// TIA Portal project "In OVO done" (V18)

(* hardware
DEVICE "S7-1200 station_1"  S7-1200 Station
   slot 0: "Rack_0"  S7-1200 Rack  Rack  V1.0
   slot 1: "plc1"  CPU 1214C DC/DC/DC  6ES7 214-1AG40-0XB0  V4.6
DEVICE "hmi1"  KTP700 Basic PN
   slot 0: "hmi1"  KTP700 Basic PN  6AV2 123-2GB03-0AX0  17.0.0.0
   slot 1: "HMI_RT_1"  KTP700 Basic PN  6AV2 123-2GB03-0AX0  17.0.0.0
   slot 5: "hmi1.IE_CP_1"  PROFINET Interface  17.0.0.0
      slot 1: "PROFINET Interface_1"  PROFINET Interface
         slot 1: "Port_1"  Port
*)

// ===== PLC "plc1"  CPU 1214C DC/DC/DC =====

VAR_GLOBAL   // PLC tag table "Default tag table"
   "System_Byte" AT %MB1 : Byte;
   "FirstScan" AT %M1.0 : Bool;
   "DiagStatusUpdate" AT %M1.1 : Bool;
   "AlwaysTRUE" AT %M1.2 : Bool;
   "AlwaysFALSE" AT %M1.3 : Bool;
   "Clock_Byte" AT %MB0 : Byte;
   "Clock_10Hz" AT %M0.0 : Bool;
   "Clock_5Hz" AT %M0.1 : Bool;
   "Clock_2.5Hz" AT %M0.2 : Bool;
   "Clock_2Hz" AT %M0.3 : Bool;
   "Clock_1.25Hz" AT %M0.4 : Bool;
   "Clock_1Hz" AT %M0.5 : Bool;
   "Clock_0.625Hz" AT %M0.6 : Bool;
   "Clock_0.5Hz" AT %M0.7 : Bool;
   "Verticaal_hot_end_Pulse" AT %Q980.0 : Bool;
   "Verticaal_hot_end_Direction" AT %Q980.1 : Bool;
END_VAR

VAR_GLOBAL   // PLC tag table "Motor"
   "motorOutput_1" AT %Q981.0 : "stepperMotorOutput";
END_VAR

VAR_GLOBAL   // PLC tag table "Valve"
   "valve1Q" AT %Q980.2 : Bool;
END_VAR

TYPE "stepperMotorInput"
   STRUCT
      axisMove : Bool;
      axisReset : Bool;
      stepOn : Bool;
      jogPlatformDown : Bool;
      jogPlatformUp : Bool;
      stateVerticalStepper : Int;   // 0 = off, 1 = needs initialization, 2 = initializing, 3 = on and initialized
      turnDistance : Real;
      shutOff : Bool;
      motorInitialize : Bool;
      motorInitialized : Bool;
      actualSpeed : Real;
      speedSelector : Int;
   END_STRUCT;
END_TYPE

TYPE "stepperMotorOutput"
   STRUCT
      TO_enable : Bool;
      Step_OFF : Bool;
   END_STRUCT;
END_TYPE

TYPE "stepperMotorSpeed"
   STRUCT
      speed300p : Real := 300.0;
      speed500p : Real := 500.0;
      speed1000p : Real := 1000.0;
      speed2000p : Real := 2000.0;
      speed3000p : Real := 3000.0;
      speed4000p : Real := 4000.0;
      speed5000p : Real := 5000.0;
      speed6000p : Real := 6000.0;
      speed7000p : Real := 7000.0;
      speed8000p : Real := 8000.0;
      speed9000p : Real := 9000.0;
      speed10000p : Real := 10000.0;
      speed11000p : Real := 11000.0;
      speed12000p : Real := 12000.0;
      speed13000p : Real := 13000.0;
      speed14000p : Real := 14000.0;
      speed15000p : Real := 15000.0;
      speed16000p : Real := 16000.0;
      speed17000p : Real := 17000.0;
      speed18000p : Real := 18000.0;
      speed19000p : Real := 19000.0;
      speed20000p : Real := 20000.0;
   END_STRUCT;
END_TYPE

TYPE "valveData"
   STRUCT
      controlHmi : Bool;
      openTime : Time;
      keepOpenHmi : Bool;
   END_STRUCT;
END_TYPE

DATA_BLOCK "openCloseCycle_DB"   // DB19
{ S7_Optimized_Access := 'TRUE' }
VERSION : 0.1
// stored: InstanceOfName openCloseCycle
"openCloseCycle"
BEGIN
END_DATA_BLOCK

DATA_BLOCK "controlStepper_DB"   // DB21
{ S7_Optimized_Access := 'TRUE' }
VERSION : 0.1
// stored: InstanceOfName controlStepper
"controlStepper"
BEGIN
END_DATA_BLOCK

// folder: Stepper/DB's

DATA_BLOCK "initVerticalStepper_DB"   // DB4
{ S7_Optimized_Access := 'TRUE' }
VERSION : 0.1
// stored: InstanceOfName initVerticalStepper
"initVerticalStepper"
BEGIN
END_DATA_BLOCK

DATA_BLOCK "stepperControlDB"   // DB8
{ S7_Optimized_Access := 'TRUE' }
VERSION : 0.1
// stored: InstanceOfName controlStepper
"controlStepper"
BEGIN
END_DATA_BLOCK

DATA_BLOCK "Motor_1"   // DB9
{ S7_Optimized_Access := 'TRUE' }
VERSION : 0.1
   VAR
      motorInput : "stepperMotorInput";
      speedPreSets : "stepperMotorSpeed";
   END_VAR
BEGIN
END_DATA_BLOCK

DATA_BLOCK "moveMotorSpeed_DB"   // DB12
{ S7_Optimized_Access := 'TRUE' }
VERSION : 0.1
// stored: InstanceOfName moveSpeedStepper
"moveSpeedStepper"
BEGIN
END_DATA_BLOCK

DATA_BLOCK "shutOffStepper_DB"   // DB16
{ S7_Optimized_Access := 'TRUE' }
VERSION : 0.1
// stored: InstanceOfName shutOffStepper
"shutOffStepper"
BEGIN
END_DATA_BLOCK

// folder: System blocks/Program resources

DATA_BLOCK "IEC_Timer_0_DB"   // DB1
{ S7_Optimized_Access := 'TRUE' }
AUTHOR : Simatic
FAMILY : IEC
NAME : IEC_TMR
VERSION : 1.0
// stored: InstanceOfName IEC_TIMER
"IEC_TIMER"
BEGIN
END_DATA_BLOCK

DATA_BLOCK "IEC_Timer_0_DB_2"   // DB14
{ S7_Optimized_Access := 'TRUE' }
AUTHOR : Simatic
FAMILY : IEC
NAME : IEC_TMR
VERSION : 1.0
// stored: InstanceOfName IEC_TIMER
"IEC_TIMER"
BEGIN
END_DATA_BLOCK

DATA_BLOCK "IEC_Timer_0_DB_4"   // DB18
{ S7_Optimized_Access := 'TRUE' }
AUTHOR : Simatic
FAMILY : IEC
NAME : IEC_TMR
VERSION : 1.0
// stored: InstanceOfName IEC_TIMER
"IEC_TIMER"
BEGIN
END_DATA_BLOCK

DATA_BLOCK "IEC_Timer_0_DB_8"   // DB24
{ S7_Optimized_Access := 'TRUE' }
AUTHOR : Simatic
FAMILY : IEC
NAME : IEC_TMR
VERSION : 1.0
// stored: InstanceOfName IEC_TIMER
"IEC_TIMER"
BEGIN
END_DATA_BLOCK

// folder: Valves/DB's

DATA_BLOCK "valvesDB"   // DB17
{ S7_Optimized_Access := 'TRUE' }
VERSION : 0.1
   VAR
      valve1 : "valveData";
   END_VAR
BEGIN
   valve1.openTime := T#500ms;
END_DATA_BLOCK

// folder: (top level)

DATA_BLOCK "VerticalHotEnd"   // DB2, Motion_DB
{ S7_Optimized_Access := 'TRUE' }
AUTHOR : SIMATIC
FAMILY : BasicMC
NAME : TO_PosAx
VERSION : 8.0
// stored: InstanceOfName TO_PositioningAxis
"TO_PositioningAxis"
BEGIN
   // Axis.EnableOutput_AddressCU = %Q981.0
   // Axis.DirectionOutputEnabledCU = TRUE
   // Axis.LengthUnit.LastDistance = -1
   // Axis.OnlinePtoModeCU = 16#0000_0002
   // Axis.SelectedChannel2EnumCU = %Q980.1
   // Axis.SelectedChannel1EnumCU = %Q980.0
   // Pulse.MinDeltaDeltaFrequencyCU = 0.004
   // Pulse.MaxDeltaDeltaFrequencyCU = 1.0E+10
   // Pulse.MinDeltaFrequencyCU = 0.005
   // Pulse.MaxDeltaFrequencyCU = 9.5E+9
   // Pulse.MinFrequencyCU = 1.0
   // Pulse.MaxFrequencyCU = 100000.0
   // Pulse.OutputSourceCU = 16#0000_0000
   // Axis.SelectPTO = 0
END_DATA_BLOCK

ORGANIZATION_BLOCK "Main"   // OB1, LAD, ProgramCycle
TITLE = "Main Program Sweep (Cycle)"
{ S7_Optimized_Access := 'TRUE' }
VERSION : 0.1
   VAR_INPUT
      Initial_Call : Bool;   // Initial call of this OB
      Remanence : Bool;   // =True, if remanent data are available
   END_VAR
BEGIN

REGION Network 1: If state is 0 but stepOn is True then change state to 1
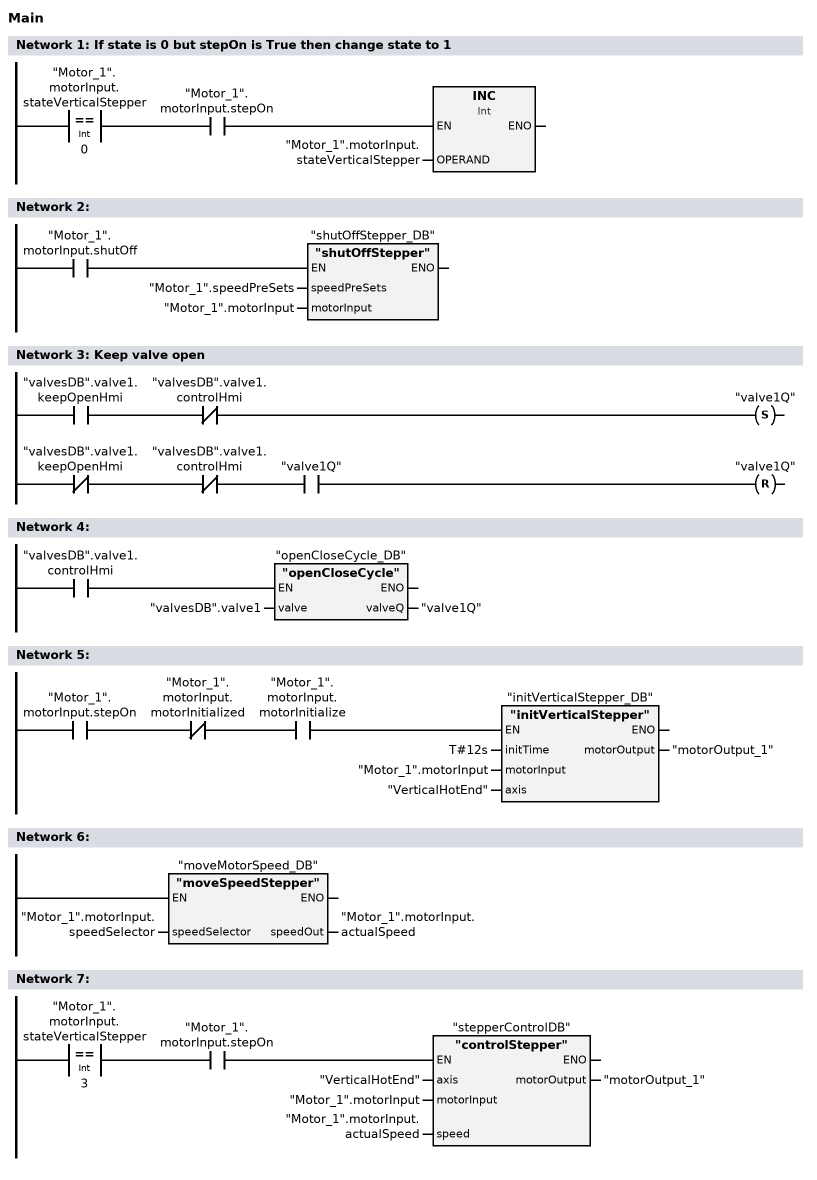
   RUNG wire#powerrail
      { S7_Templates := "SrcType := Int" } EQ_Contact(in1 := "Motor_1".motorInput.stateVerticalStepper, in2 := 0)
      Contact( "Motor_1".motorInput.stepOn )
      { S7_Templates := "DestType := Int" } Inc( "Motor_1".motorInput.stateVerticalStepper )
   END_RUNG
   // the same network as SCL:
   IF ("Motor_1".motorInput.stateVerticalStepper = 0) AND "Motor_1".motorInput.stepOn THEN
       "Motor_1".motorInput.stateVerticalStepper := "Motor_1".motorInput.stateVerticalStepper + 1;
   END_IF;
END_REGION

REGION Network 2
   RUNG wire#powerrail
      Contact( "Motor_1".motorInput.shutOff )
      "shutOffStepper_DB"(speedPreSets := "Motor_1".speedPreSets, motorInput := "Motor_1".motorInput)
   END_RUNG
   // the same network as SCL:
   IF "Motor_1".motorInput.shutOff THEN
       "shutOffStepper_DB"(speedPreSets := "Motor_1".speedPreSets, motorInput := "Motor_1".motorInput);   // "shutOffStepper"
   END_IF;
END_REGION

REGION Network 3: Keep valve open
   RUNG wire#powerrail
      Contact( "valvesDB".valve1.keepOpenHmi )
      I_Contact( "valvesDB".valve1.controlHmi )
      S_Coil( "valve1Q" )
   END_RUNG
   RUNG wire#powerrail
      I_Contact( "valvesDB".valve1.keepOpenHmi )
      I_Contact( "valvesDB".valve1.controlHmi )
      Contact( "valve1Q" )
      R_Coil( "valve1Q" )
   END_RUNG
   // the same network as SCL:
   IF "valvesDB".valve1.keepOpenHmi AND NOT "valvesDB".valve1.controlHmi THEN "valve1Q" := TRUE; END_IF;
   IF NOT "valvesDB".valve1.keepOpenHmi AND NOT "valvesDB".valve1.controlHmi AND "valve1Q" THEN
       "valve1Q" := FALSE;
   END_IF;
END_REGION

REGION Network 4
   RUNG wire#powerrail
      Contact( "valvesDB".valve1.controlHmi )
      "openCloseCycle_DB"(valve := "valvesDB".valve1, valveQ => "valve1Q")
   END_RUNG
   // the same network as SCL:
   IF "valvesDB".valve1.controlHmi THEN
       "openCloseCycle_DB"(valve := "valvesDB".valve1, valveQ => "valve1Q");   // "openCloseCycle"
   END_IF;
END_REGION

REGION Network 5
   RUNG wire#powerrail
      Contact( "Motor_1".motorInput.stepOn )
      I_Contact( "Motor_1".motorInput.motorInitialized )
      Contact( "Motor_1".motorInput.motorInitialize )
      "initVerticalStepper_DB"(initTime := T#12s, motorInput := "Motor_1".motorInput, axis := "VerticalHotEnd", motorOutput => "motorOutput_1")
   END_RUNG
   // the same network as SCL:
   IF "Motor_1".motorInput.stepOn AND NOT "Motor_1".motorInput.motorInitialized AND "Motor_1".motorInput.motorInitialize THEN
       "initVerticalStepper_DB"(initTime := T#12s,   // "initVerticalStepper"
                               motorInput := "Motor_1".motorInput,
                               axis := "VerticalHotEnd",
                               motorOutput => "motorOutput_1");
   END_IF;
END_REGION

REGION Network 6
   RUNG wire#powerrail
      "moveMotorSpeed_DB"(speedSelector := "Motor_1".motorInput.speedSelector, speedOut => "Motor_1".motorInput.actualSpeed)
   END_RUNG
   // the same network as SCL:
   "moveMotorSpeed_DB"(speedSelector := "Motor_1".motorInput.speedSelector,   // "moveSpeedStepper"
                       speedOut => "Motor_1".motorInput.actualSpeed);
END_REGION

REGION Network 7
   RUNG wire#powerrail
      { S7_Templates := "SrcType := Int" } EQ_Contact(in1 := "Motor_1".motorInput.stateVerticalStepper, in2 := 3)
      Contact( "Motor_1".motorInput.stepOn )
      "stepperControlDB"(axis := "VerticalHotEnd", motorInput := "Motor_1".motorInput, speed := "Motor_1".motorInput.actualSpeed, motorOutput => "motorOutput_1")
   END_RUNG
   // the same network as SCL:
   IF ("Motor_1".motorInput.stateVerticalStepper = 3) AND "Motor_1".motorInput.stepOn THEN
       "stepperControlDB"(axis := "VerticalHotEnd",   // "controlStepper"
                          motorInput := "Motor_1".motorInput,
                          speed := "Motor_1".motorInput.actualSpeed,
                          motorOutput => "motorOutput_1");
   END_IF;
END_REGION
END_ORGANIZATION_BLOCK

// folder: Stepper

FUNCTION_BLOCK "controlStepper"   // FB1, LAD
{ S7_Optimized_Access := 'TRUE' }
VERSION : 0.1
   VAR_INPUT
      axis : TO_PositioningAxis;
      motorInput : "stepperMotorInput";
      speed : Int;
   END_VAR
   VAR_OUTPUT
      motorOutput : "stepperMotorOutput";
   END_VAR
BEGIN

REGION Network 1: enable motor
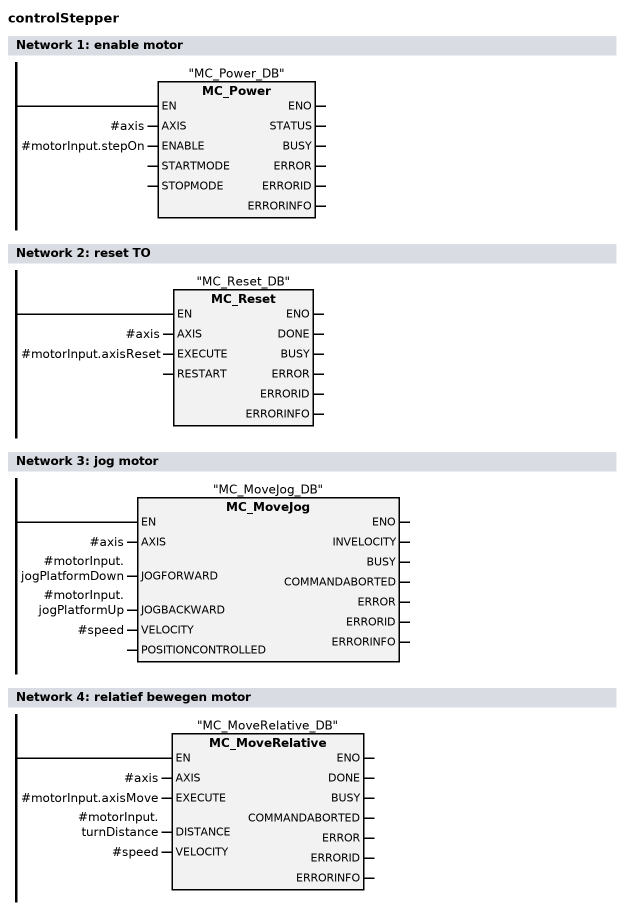
   "MC_Power_DB"(Axis := #axis, Enable := #motorInput.stepOn);   // MC_Power
END_REGION

REGION Network 2: reset TO
   "MC_Reset_DB"(Axis := #axis, Execute := #motorInput.axisReset);   // MC_Reset
END_REGION

REGION Network 3: jog motor
   "MC_MoveJog_DB"(Axis := #axis,   // MC_MoveJog
                   JogForward := #motorInput.jogPlatformDown,
                   JogBackward := #motorInput.jogPlatformUp,
                   Velocity := #speed);
END_REGION

REGION Network 4: relatief bewegen motor
   "MC_MoveRelative_DB"(Axis := #axis,   // MC_MoveRelative
                        Execute := #motorInput.axisMove,
                        Distance := #motorInput.turnDistance,
                        Velocity := #speed);
END_REGION
END_FUNCTION_BLOCK

FUNCTION_BLOCK "initVerticalStepper"   // FB2, LAD
TITLE = Initialize vertical stepper
{ S7_Optimized_Access := 'TRUE' }
VERSION : 0.1
   VAR_INPUT
      initTime : Time;
   END_VAR
   VAR_OUTPUT
      motorOutput : "stepperMotorOutput";
   END_VAR
   VAR_IN_OUT
      motorInput : "stepperMotorInput";
      axis : TO_PositioningAxis;
   END_VAR
BEGIN

REGION Network 1: Turn platform into screw thread and set state to initializing. Set a timer and after that reset the initialize tag and set state to "on and initialized"
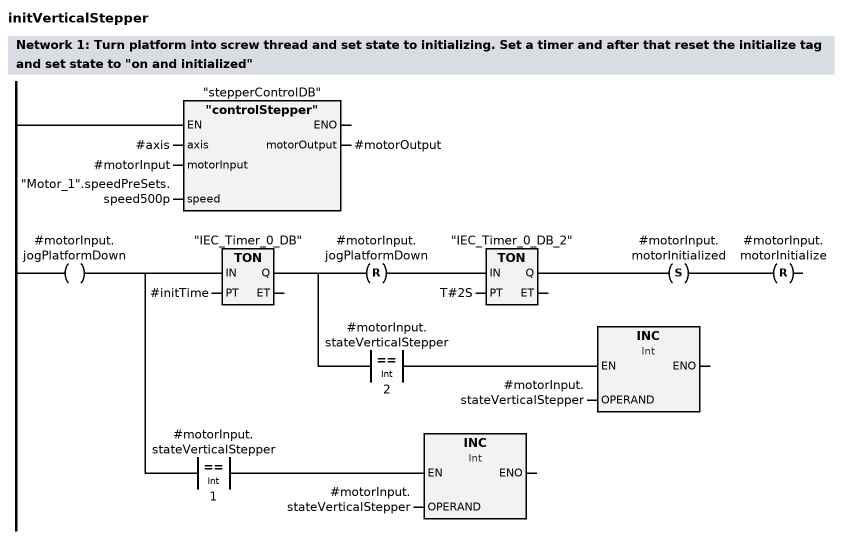
   "stepperControlDB"(axis := #axis,   // "controlStepper"
                      motorInput := #motorInput,
                      speed := "Motor_1".speedPreSets.speed500p,
                      motorOutput => #motorOutput);
   #motorInput.jogPlatformDown := TRUE;
   "IEC_Timer_0_DB".TON(IN := TRUE, PT := #initTime);
   IF "IEC_Timer_0_DB".Q THEN #motorInput.jogPlatformDown := FALSE; END_IF;
   "IEC_Timer_0_DB_2".TON(IN := "IEC_Timer_0_DB".Q, PT := T#2S);
   IF "IEC_Timer_0_DB_2".Q THEN
       #motorInput.motorInitialized := TRUE;
       #motorInput.motorInitialize := FALSE;
   END_IF;
   IF "IEC_Timer_0_DB".Q AND (#motorInput.stateVerticalStepper = 2) THEN
       #motorInput.stateVerticalStepper := #motorInput.stateVerticalStepper + 1;
   END_IF;
   IF #motorInput.stateVerticalStepper = 1 THEN
       #motorInput.stateVerticalStepper := #motorInput.stateVerticalStepper + 1;
   END_IF;
END_REGION
END_FUNCTION_BLOCK

FUNCTION_BLOCK "moveSpeedStepper"   // FB4, LAD
{ S7_Optimized_Access := 'TRUE' }
VERSION : 0.1
   VAR_INPUT
      speedSelector : Int;
   END_VAR
   VAR_OUTPUT
      speedOut : Real;
   END_VAR
   VAR
      speeds : "stepperMotorSpeed";
   END_VAR
BEGIN

REGION Network 1
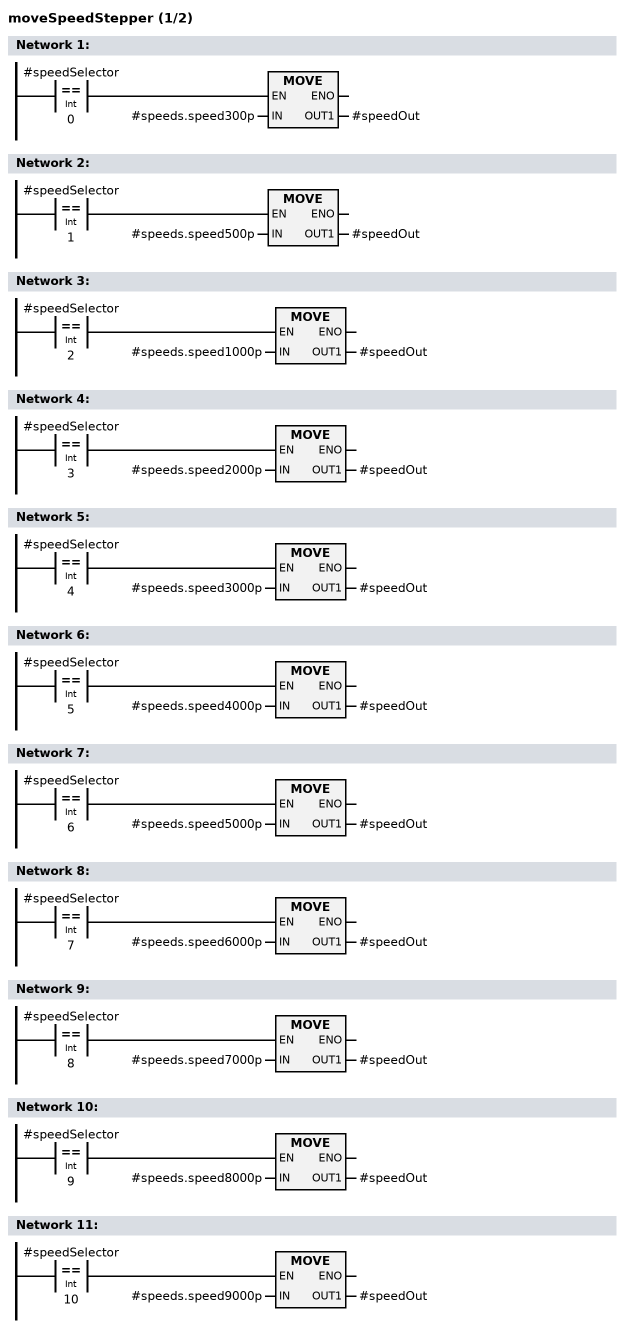
   RUNG wire#powerrail
      { S7_Templates := "SrcType := Int" } EQ_Contact(in1 := #speedSelector, in2 := 0)
      Move(in := #speeds.speed300p, out1 => #speedOut)
   END_RUNG
   // the same network as SCL:
   IF #speedSelector = 0 THEN #speedOut := #speeds.speed300p; END_IF;
END_REGION

REGION Network 2
   RUNG wire#powerrail
      { S7_Templates := "SrcType := Int" } EQ_Contact(in1 := #speedSelector, in2 := 1)
      Move(in := #speeds.speed500p, out1 => #speedOut)
   END_RUNG
   // the same network as SCL:
   IF #speedSelector = 1 THEN #speedOut := #speeds.speed500p; END_IF;
END_REGION

REGION Network 3
   RUNG wire#powerrail
      { S7_Templates := "SrcType := Int" } EQ_Contact(in1 := #speedSelector, in2 := 2)
      Move(in := #speeds.speed1000p, out1 => #speedOut)
   END_RUNG
   // the same network as SCL:
   IF #speedSelector = 2 THEN #speedOut := #speeds.speed1000p; END_IF;
END_REGION

REGION Network 4
   RUNG wire#powerrail
      { S7_Templates := "SrcType := Int" } EQ_Contact(in1 := #speedSelector, in2 := 3)
      Move(in := #speeds.speed2000p, out1 => #speedOut)
   END_RUNG
   // the same network as SCL:
   IF #speedSelector = 3 THEN #speedOut := #speeds.speed2000p; END_IF;
END_REGION

REGION Network 5
   RUNG wire#powerrail
      { S7_Templates := "SrcType := Int" } EQ_Contact(in1 := #speedSelector, in2 := 4)
      Move(in := #speeds.speed3000p, out1 => #speedOut)
   END_RUNG
   // the same network as SCL:
   IF #speedSelector = 4 THEN #speedOut := #speeds.speed3000p; END_IF;
END_REGION

REGION Network 6
   RUNG wire#powerrail
      { S7_Templates := "SrcType := Int" } EQ_Contact(in1 := #speedSelector, in2 := 5)
      Move(in := #speeds.speed4000p, out1 => #speedOut)
   END_RUNG
   // the same network as SCL:
   IF #speedSelector = 5 THEN #speedOut := #speeds.speed4000p; END_IF;
END_REGION

REGION Network 7
   RUNG wire#powerrail
      { S7_Templates := "SrcType := Int" } EQ_Contact(in1 := #speedSelector, in2 := 6)
      Move(in := #speeds.speed5000p, out1 => #speedOut)
   END_RUNG
   // the same network as SCL:
   IF #speedSelector = 6 THEN #speedOut := #speeds.speed5000p; END_IF;
END_REGION

REGION Network 8
   RUNG wire#powerrail
      { S7_Templates := "SrcType := Int" } EQ_Contact(in1 := #speedSelector, in2 := 7)
      Move(in := #speeds.speed6000p, out1 => #speedOut)
   END_RUNG
   // the same network as SCL:
   IF #speedSelector = 7 THEN #speedOut := #speeds.speed6000p; END_IF;
END_REGION

REGION Network 9
   RUNG wire#powerrail
      { S7_Templates := "SrcType := Int" } EQ_Contact(in1 := #speedSelector, in2 := 8)
      Move(in := #speeds.speed7000p, out1 => #speedOut)
   END_RUNG
   // the same network as SCL:
   IF #speedSelector = 8 THEN #speedOut := #speeds.speed7000p; END_IF;
END_REGION

REGION Network 10
   RUNG wire#powerrail
      { S7_Templates := "SrcType := Int" } EQ_Contact(in1 := #speedSelector, in2 := 9)
      Move(in := #speeds.speed8000p, out1 => #speedOut)
   END_RUNG
   // the same network as SCL:
   IF #speedSelector = 9 THEN #speedOut := #speeds.speed8000p; END_IF;
END_REGION

REGION Network 11
   RUNG wire#powerrail
      { S7_Templates := "SrcType := Int" } EQ_Contact(in1 := #speedSelector, in2 := 10)
      Move(in := #speeds.speed9000p, out1 => #speedOut)
   END_RUNG
   // the same network as SCL:
   IF #speedSelector = 10 THEN #speedOut := #speeds.speed9000p; END_IF;
END_REGION

REGION Network 12
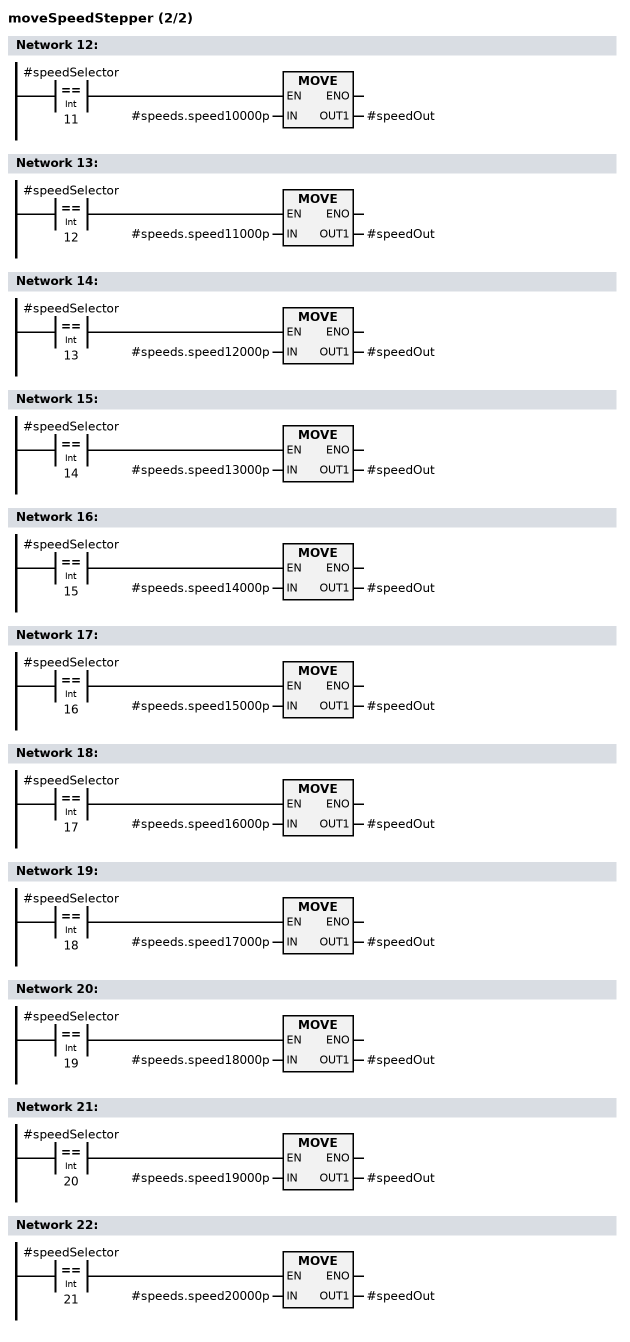
   RUNG wire#powerrail
      { S7_Templates := "SrcType := Int" } EQ_Contact(in1 := #speedSelector, in2 := 11)
      Move(in := #speeds.speed10000p, out1 => #speedOut)
   END_RUNG
   // the same network as SCL:
   IF #speedSelector = 11 THEN #speedOut := #speeds.speed10000p; END_IF;
END_REGION

REGION Network 13
   RUNG wire#powerrail
      { S7_Templates := "SrcType := Int" } EQ_Contact(in1 := #speedSelector, in2 := 12)
      Move(in := #speeds.speed11000p, out1 => #speedOut)
   END_RUNG
   // the same network as SCL:
   IF #speedSelector = 12 THEN #speedOut := #speeds.speed11000p; END_IF;
END_REGION

REGION Network 14
   RUNG wire#powerrail
      { S7_Templates := "SrcType := Int" } EQ_Contact(in1 := #speedSelector, in2 := 13)
      Move(in := #speeds.speed12000p, out1 => #speedOut)
   END_RUNG
   // the same network as SCL:
   IF #speedSelector = 13 THEN #speedOut := #speeds.speed12000p; END_IF;
END_REGION

REGION Network 15
   RUNG wire#powerrail
      { S7_Templates := "SrcType := Int" } EQ_Contact(in1 := #speedSelector, in2 := 14)
      Move(in := #speeds.speed13000p, out1 => #speedOut)
   END_RUNG
   // the same network as SCL:
   IF #speedSelector = 14 THEN #speedOut := #speeds.speed13000p; END_IF;
END_REGION

REGION Network 16
   RUNG wire#powerrail
      { S7_Templates := "SrcType := Int" } EQ_Contact(in1 := #speedSelector, in2 := 15)
      Move(in := #speeds.speed14000p, out1 => #speedOut)
   END_RUNG
   // the same network as SCL:
   IF #speedSelector = 15 THEN #speedOut := #speeds.speed14000p; END_IF;
END_REGION

REGION Network 17
   RUNG wire#powerrail
      { S7_Templates := "SrcType := Int" } EQ_Contact(in1 := #speedSelector, in2 := 16)
      Move(in := #speeds.speed15000p, out1 => #speedOut)
   END_RUNG
   // the same network as SCL:
   IF #speedSelector = 16 THEN #speedOut := #speeds.speed15000p; END_IF;
END_REGION

REGION Network 18
   RUNG wire#powerrail
      { S7_Templates := "SrcType := Int" } EQ_Contact(in1 := #speedSelector, in2 := 17)
      Move(in := #speeds.speed16000p, out1 => #speedOut)
   END_RUNG
   // the same network as SCL:
   IF #speedSelector = 17 THEN #speedOut := #speeds.speed16000p; END_IF;
END_REGION

REGION Network 19
   RUNG wire#powerrail
      { S7_Templates := "SrcType := Int" } EQ_Contact(in1 := #speedSelector, in2 := 18)
      Move(in := #speeds.speed17000p, out1 => #speedOut)
   END_RUNG
   // the same network as SCL:
   IF #speedSelector = 18 THEN #speedOut := #speeds.speed17000p; END_IF;
END_REGION

REGION Network 20
   RUNG wire#powerrail
      { S7_Templates := "SrcType := Int" } EQ_Contact(in1 := #speedSelector, in2 := 19)
      Move(in := #speeds.speed18000p, out1 => #speedOut)
   END_RUNG
   // the same network as SCL:
   IF #speedSelector = 19 THEN #speedOut := #speeds.speed18000p; END_IF;
END_REGION

REGION Network 21
   RUNG wire#powerrail
      { S7_Templates := "SrcType := Int" } EQ_Contact(in1 := #speedSelector, in2 := 20)
      Move(in := #speeds.speed19000p, out1 => #speedOut)
   END_RUNG
   // the same network as SCL:
   IF #speedSelector = 20 THEN #speedOut := #speeds.speed19000p; END_IF;
END_REGION

REGION Network 22
   RUNG wire#powerrail
      { S7_Templates := "SrcType := Int" } EQ_Contact(in1 := #speedSelector, in2 := 21)
      Move(in := #speeds.speed20000p, out1 => #speedOut)
   END_RUNG
   // the same network as SCL:
   IF #speedSelector = 21 THEN #speedOut := #speeds.speed20000p; END_IF;
END_REGION
END_FUNCTION_BLOCK

FUNCTION_BLOCK "shutOffStepper"   // FB5, LAD
{ S7_Optimized_Access := 'TRUE' }
VERSION : 0.1
   VAR_INPUT
      speedPreSets : "stepperMotorSpeed";
   END_VAR
   VAR_IN_OUT
      motorInput : "stepperMotorInput";
   END_VAR
BEGIN

REGION Network 1
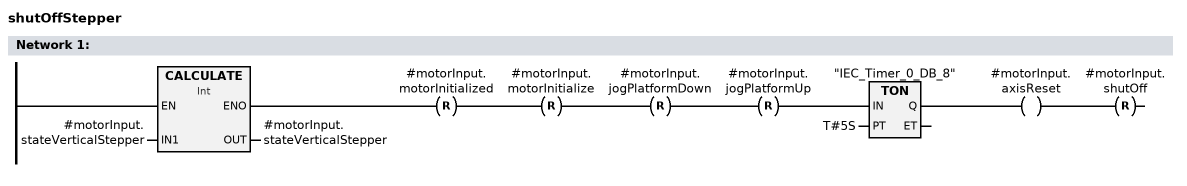
   #motorInput.stateVerticalStepper := #motorInput.stateVerticalStepper-#motorInput.stateVerticalStepper;
   #motorInput.motorInitialized := FALSE;
   #motorInput.motorInitialize := FALSE;
   #motorInput.jogPlatformDown := FALSE;
   #motorInput.jogPlatformUp := FALSE;
   "IEC_Timer_0_DB_8".TON(IN := TRUE, PT := T#5S);
   #motorInput.axisReset := "IEC_Timer_0_DB_8".Q;
   IF "IEC_Timer_0_DB_8".Q THEN #motorInput.shutOff := FALSE; END_IF;
END_REGION
END_FUNCTION_BLOCK

// folder: Valves

FUNCTION_BLOCK "openCloseCycle"   // FB7, LAD
{ S7_Optimized_Access := 'TRUE' }
VERSION : 0.1
   VAR_OUTPUT
      valveQ : Bool;
   END_VAR
   VAR_IN_OUT
      valve : "valveData";
   END_VAR
   VAR_TEMP   // added for the SCL form of the ladder/FBD networks
      _w1 : Bool;
   END_VAR
BEGIN

REGION Network 1
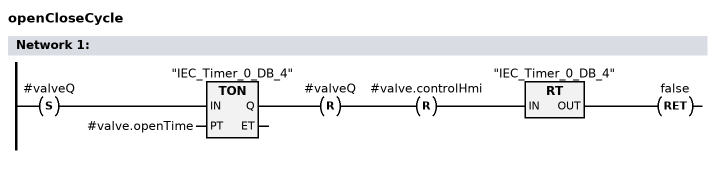
   #valveQ := TRUE;
   "IEC_Timer_0_DB_4".TON(IN := TRUE, PT := #valve.openTime);
   IF "IEC_Timer_0_DB_4".Q THEN
       #valveQ := FALSE;
       #valve.controlHmi := FALSE;
   END_IF;
   #_w1 := "IEC_Timer_0_DB_4".Q;
   IF #_w1 THEN
       RESET_TIMER("IEC_Timer_0_DB_4");
       ENO := false;
       RETURN;
   END_IF;
END_REGION
END_FUNCTION_BLOCK

(* ===== HMI "HMI_RT_1" =====
system functions are stored by id; their names below are inferred from use
connection "HMI_Connection_1": ETHERNET, SMART_S7_1200_OMS

HMI tags "Default tag table"
   "Tag_ScreenNumber" : UInt, internal
   "valveEggs_1" : Bool = PLC valve1Q AT %Q980.2, 100 ms
   "valvesDB_valve1_controlHmi" : Bool = PLC valvesDB.valve1.controlHmi, 100 ms
   "valvesDB_valve1_openTime" : Time = PLC valvesDB.valve1.openTime, 100 ms
   "valvesDB_valve1_keepOpenHmi" : Bool = PLC valvesDB.valve1.keepOpenHmi, 100 ms

HMI tags "Stepper_motor"
   "Motor_Q_1" : stepperMotorOutput = PLC motorOutput_1 AT %Q981.0, 100 ms
   "Motor_I_1" : stepperMotorInput = PLC Motor_1.motorInput AT %DB1.DBW0, 100 ms
   "Verticaal_hot_end_Direction" : Bool = PLC Verticaal_hot_end_Direction AT %Q980.1, 1 s
   "Verticaal_hot_end_Pulse" : Bool = PLC Verticaal_hot_end_Pulse AT %Q980.0, 1 s

Template "Template_1" 800x480
   Button "Template_Button_3" at 316,429 size 71x50; TextOff 'Text'
   Button "Exit" at 714,429 size 71x50; TextOff 'Exit'; PictureOff "ExitRuntime_KTP700_Basic_PN_TR"; PictureOn "ExitRuntime_KTP700_Basic_PN_TR"
      on Release: StopRuntime(0)
   Button "Template_Button" at 614,429 size 71x50; TextOff 'Text'
   Button "Template_Button_1" at 514,429 size 71x50; TextOff 'Text'
   Button "Template_Button_2" at 414,429 size 71x50; TextOff 'Text'
   Button "Template_Button_4" at 214,429 size 71x50; TextOff 'Text'
   Button "Alarms" at 114,429 size 71x50; TextOff 'Alarms'; PictureOff "AlarmDisplay_KTP700_Basic_PN_TR"; PictureOn "AlarmDisplay_KTP700_Basic_PN_TR"
      on Release: function_ef3f5d25("Alarm window_Unacknowledged", -1)
   Button "Start screen" at 14,429 size 71x50; TextOff 'Start screen'; PictureOff "NavigateHome_KTP700_Basic_PN_TR"; PictureOn "NavigateHome_KTP700_Basic_PN_TR"
      on Release: ActivateScreen("Root screen", 0)
   SymbolicIOField "Symbolic_IO_Field_Screen" at 93,9 size 600x33; TextOff '0'; TextOn '1'; TextList "TextList_ScreenNames"
      ProcessValue <- "Tag_ScreenNumber"
      on Change: ActivateScreenByNumber("Tag_ScreenNumber", 0)
   DateTimeField "HmiScreenItemData" at 695,25 size 105x25
   DateTimeField "HmiScreenItemData_1" at 695,0 size 105x25
   GraphicView "Logo" at 0,0 size 91x51; Picture "In+Ovo+logo_2"

screen "Root screen" 800x480, template "Template_1"
   on GenerateScreen: SetTag("Tag_ScreenNumber", 1)
   Button "Button_3" at 404,264 size 148x64; TextOff 'Start glueing'; PictureOff "Graphic_2"
      on Press: SetBit("valvesDB_valve1_controlHmi"); ResetBit("valvesDB_valve1_keepOpenHmi"); function_b14e0dd5("valvesDB_valve1_controlHmi", 0)
   GraphicView "Graphic view_1" at 334,141 size 133x70; Picture "Graphic_1"
   TextField "Text field_1" at 302,107 size 197x23; Text 'Vertical stepper motors'
   Circle "Circle_1" at 445,224 size 32x32
      Appearance <- "stateVerticalStepper"
   Switch "Switch_1" at 329,224 size 109x32; CaptionText 'Switch'; TextOff 'OFF'; TextOn 'ON'
      ProcessValue <- "stepOn"
      on SwitchOff: SetBit("shutOff")
   Button "Button_1" at 245,264 size 148x64; TextOff 'Initialize'
      on Press: SetBit("motorInitialize")
   Button "Button_2" at 245,336 size 307x32; TextOff 'Manual control/settings'; TextOn 'Manual control'
      on Click: ActivateScreen("Manual control", 0)
   GraphicView "Graphic view_2" at 570,118 size 183x250; Picture "580b57fbd9996e24bc43c108"
   GraphicView "Graphic view_3" at 18,129 size 225x239; Picture "308-3089671_baby-chicken-free-png-image-chick-transparent-png"

screen "Manual control" 800x480, template "Template_1"
   Button "Button_2" at 226,210 size 109x64; TextOff 'Down'
      on Release: ResetBit("jogPlatformDown")
      on Press: SetBit("jogPlatformDown"); ResetBit("jogPlatformUp")
   Button "Button_3" at 226,136 size 109x64; TextOff 'Up'
      on Release: ResetBit("jogPlatformUp")
      on Press: SetBit("jogPlatformUp"); ResetBit("jogPlatformDown")
   IOField "I/O field_1" at 593,168 size 109x32; FormatPattern s999999999.999
      ProcessValue <- "turnDistance"
   Button "Button_4" at 227,284 size 109x64; TextOff 'Move'
      on Release: ResetBit("axisMove")
      on Press: SetBit("axisMove")
   TextField "Text field_3" at 238,105 size 86x23; Text 'Jog/move'
   TextField "Text field_4" at 345,105 size 112x23; Text 'Valve control'
   TextField "Text field_2" at 587,136 size 121x23; Text 'Move distance'
   IOField "I/O field_2" at 593,242 size 109x32; FormatPattern s999999999.999
      ProcessValue <- "actualSpeed"
   Button "Button_5" at 466,136 size 109x64; TextOff '+'; PictureOff "Graphic_2"
      on Press: function_dd21b452("speedSelector", 1)
   Button "Button_6" at 466,210 size 109x64; TextOff '-'; PictureOff "Graphic_3"
      on Press: function_b9b71300("speedSelector", 1)
   TextField "Text field_5" at 593,210 size 109x32; Text 'Jog speed'
   Button "Button_1" at 226,359 size 349x32; TextOff 'Root screen'
      on Click: ActivateScreen("Root screen", 0)
   GraphicView "Graphic view_1" at 52,140 size 133x70; Picture "Graphic_1"
   TextField "Text field_1" at 20,106 size 197x23; Text 'Vertical stepper motors'
   Circle "Circle_1" at 161,223 size 32x32
      Appearance <- "stateVerticalStepper"
   Switch "Switch_1" at 45,223 size 109x32; TextOn 'ON'; CaptionText 'Switch'; TextOff 'OFF'
      on SwitchOff: SetBit("shutOff")
      ProcessValue <- "stepOn"
   Button "Button_7" at 45,263 size 148x64; TextOff 'Initialize'
      on Press: SetBit("motorInitialize")
   TextField "Text field_6" at 468,105 size 106x23; Text 'Motor speed'
   Switch "Switch_4" at 346,210 size 109x64; TextOn 'Open'; CaptionText 'Switch'; TextOff 'Closed'
      on SwitchOn: ResetBit("valvesDB_valve1_controlHmi")
      ProcessValue <- "valvesDB_valve1_keepOpenHmi"
   IOField "I/O field_3" at 593,316 size 109x32; FormatPattern s9999999999
      ProcessValue <- "valvesDB_valve1_openTime"
   TextField "Text field_9" at 579,284 size 137x23; Text 'Valve open time'
   Button "Button_9" at 346,136 size 109x64; TextOff 'Open'
      on Press: SetBit("valvesDB_valve1_controlHmi"); ResetBit("valvesDB_valve1_keepOpenHmi")
*)